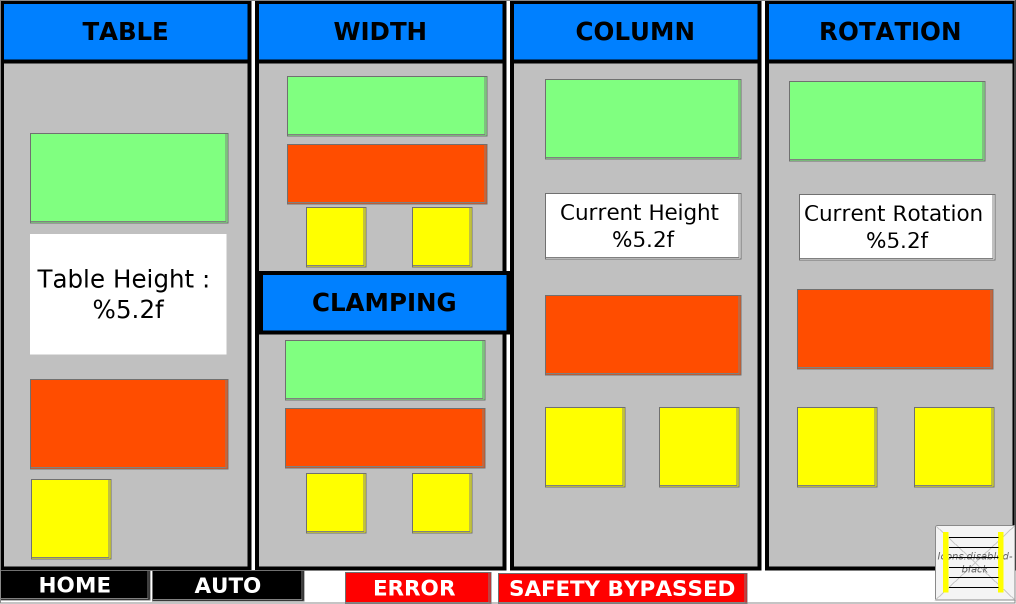
VISUALIZATION manualBypassedScreen  // 1016x604
    Group (0,0 1016x570)
        Rectangle (255,0 251x570)
        Rectangle (510,0 251x570)
        Rectangle (765,0 251x570)
        Rectangle (0,0 251x570)
    Button (545,79 196x80), image: Icons.up-black
        OnMouseDown: execute { manual.eColumnState := 1; }
        OnMouseUp: execute { manual.eColumnState := 0; }
    Button (545,295 196x80), image: Icons.down-black
        OnMouseDown: execute { manual.eColumnState := 2; }
        OnMouseUp: execute { manual.eColumnState := 0; }
    Button (797,289 196x80), image: Icons.rotate-ccw-black
        OnMouseDown: execute { manual.eRotationState := 1; }
        OnMouseUp: execute { manual.eRotationState := 0; }
    Button (789,81 196x80), image: Icons.rotate-ccw-black0
        OnMouseDown: execute { manual.eRotationState := 2; }
        OnMouseUp: execute { manual.eRotationState := 0; }
    Button (545,407 80x80), image: Icons.home-black
        OnMouseDown: execute { manual.eColumnState := 4; }
    Button (797,407 80x80), image: Icons.home-black
        OnMouseDown: execute { manual.eRotationState := 4; }
    Button (659,407 80x80), image: Icons.reset-black
        OnMouseDown: execute { manual.eColumnState := 3; }
    Button (914,407 80x80), image: Icons.reset-black
        OnMouseDown: execute { manual.eRotationState := 3; }
    Button (412,473 60x60), image: Icons.reset-black
        OnMouseDown: execute { manual.eClampingState := 3; }
    Button (287,76 200x60), image: Icons.width-in-black
        OnMouseDown: execute { manual.eWidthState := 1; }
        OnMouseUp: execute { manual.eWidthState := 0; }
    Button (287,144 200x60), image: Icons.width-out-black
        OnMouseDown: execute { manual.eWidthState := 2; }
        OnMouseUp: execute { manual.eWidthState := 0; }
    Button (285,340 200x60), image: Icons.Unclamp-black
        OnMouseDown: execute { manual.eClampingState := 1; }
        OnMouseUp: execute { manual.eClampingState := 0; }
    Button (285,408 200x60), image: Icons.clamp-black
        OnMouseDown: execute { manual.eClampingState := 2; }
        OnMouseUp: execute { manual.eClampingState := 0; }
    Button (306,473 60x60), image: Icons.home-black
        OnMouseDown: execute { manual.eClampingState := 4; }
    Button (306,207 60x60), image: Icons.home-black
        OnMouseDown: execute { manual.eWidthState := 4; }
    Button (412,207 60x60), image: Icons.reset-black
        OnMouseDown: execute { manual.eWidthState := 3; }
    Button (30,379 198x90), image: Icons.down-black
        OnMouseDown: execute { manual.eTableState := 2; }
        OnMouseUp: execute { manual.eTableState := 0; }
    RoundedRectangle (0,0 251x63), "TABLE", colour toggle: manual.bTableMoveStatus
    RoundedRectangle (255,0 251x63), "WIDTH", colour toggle: manual.bWidthMoveStatus
    RoundedRectangle (510,0 251x63), "COLUMN", colour toggle: manual.bColumnMoveStatus
    RoundedRectangle (765,0 251x63), "ROTATION", colour toggle: manual.bRotationMoveStatus
    Button (30,133 198x90), image: Icons.up-black
        OnMouseDown: execute { manual.eTableState := 1; }
        OnMouseUp: execute { manual.eTableState := 0; }
    RoundedRectangle (30,234 196x120), "Table Height : %5.2f", text variable: GVL_ignition.fTableHeight
    Button (545,193 196x66), "Current Height %5.2f", text variable: GVL_ignition.fColumnHeight
    RoundedRectangle (259,271 251x63), "CLAMPING", colour toggle: manual.bClampingMoveStatus
    Button (0,570 150x30), "HOME"
        OnMouseDown: change screen: mainScreen
        OnMouseDown: execute { GVL_machine.nPageIndex := 0; }
    Button (152,570 152x31), "AUTO"
        OnMouseDown: change screen: eflexScreen
        OnMouseDown: execute { GVL_machine.nPageIndex := 10; }
    Button (799,194 196x66), "Current Rotation %5.2f", text variable: GVL_ignition.fRotationDistance
    Button (31,479 80x80), image: Icons.home-black
        OnMouseDown: execute { manual.eTableState := 4; }
    Image (935,525 80x75), invisible if: MAIN.bHideLtCurtainDisable, image: Icons.disabled-black
    Group (943,532 60x60), invisible if: GVL_machine.bSafetyBypass
        toggle GVL_machine.bMuteSafety
        Rectangle (0,0 5x60)
        Rectangle (55,0 5x60)
        Line (6,5) (55,5)
        Line (6,15) (55,15)
        Line (6,25) (55,25)
        Line (6,35) (55,35)
        Line (6,45) (55,45)
        Line (6,55) (55,55)
    Button (498,573 249x31), "SAFETY BYPASSED", invisible if: NOT GVL_machine.bSafetyBypass
        OnMouseDown: change screen: safetyDisableWarning
    Button (345,572 146x32), "ERROR", invisible if: NOT GVL_machine.bDispErrorIcon
        OnMouseDown: change screen: errorScreen
END_VISUALIZATION

(* stored: Version 1.1.0.1, ProductVersion 3.1.4024.13
   Visu manualBypassedScreen: Id {7372f360-6185-47c7-80ce-482ad0b0e7bf} *)
